FUNCTION_BLOCK treinrit
VAR_INPUT
    Start : BOOL;
    TravelTime : TIME;
END_VAR

VAR_OUTPUT
    Arrived : BOOL := FALSE;
END_VAR

VAR
END_VAR

IF Start AND NOT gvl.InternalStart THEN
    gvl.InternalStart := TRUE;
    Arrived := FALSE;
    gvl.Timer(IN := TRUE, PT := TravelTime);
END_IF;

gvl.Timer(IN := gvl.Timer.IN, PT := TravelTime);


IF gvl.Timer.Q THEN
    Arrived := TRUE;
    gvl.Timer(IN := FALSE);
    gvl.InternalStart := FALSE;
END_IF;

END_FUNCTION_BLOCK

(* stored: Version 1.1.0.1, ProductVersion 3.1.4024.15
   POU treinrit: Id {1113fe9e-cd66-49f9-a801-011964240413}, SpecialFunc None *)
